FUNCTION_BLOCK FB_EZylinder
VAR_INPUT
	bgate : BOOL;
	berror : BOOL;
END_VAR
VAR_OUTPUT
	bR1 : BOOL;
	bR2 : BOOL;
END_VAR
VAR
END_VAR


bR1 := bgate;
bR2 := NOT bgate;

IF berror THEN
	bR1 := FALSE;
	bR2 := FALSE;
	
END_IF

END_FUNCTION_BLOCK

(* stored: Version 1.1.0.1, ProductVersion 3.1.4024.15
   POU FB_EZylinder: Id {e63bf942-b98e-47d4-9691-d62e1cea7af4}, SpecialFunc None *)
